// TwinCAT 3 PLC project M1L1_PLC
// ProgramVersion: 3.1.4020.5
// libraries:
//   LCLS General, * (SLAC)
//   Tc2_MC2, * (Beckhoff Automation GmbH)
//   Tc2_SerialCom, * (Beckhoff Automation GmbH)
//   Tc2_Standard, * (Beckhoff Automation GmbH)
//   Tc2_System, * (Beckhoff Automation GmbH)
//   Tc2_Utilities, * (Beckhoff Automation GmbH)
//   Tc3_Module, * (Beckhoff Automation GmbH)
//   lcls-twincat-motion,1.1.0,SLAC
// project tree:
//   Common/POUs/Helpers/ FB_PI_E621_SerialDriver.TcPOU (not stored), FB_PI_E621_SerialTransaction.TcPOU (not stored)
//   DUTs/ ST_PiezoAxis.TcDUT (not stored)
//   GVLs/ GVL_SerialIO.TcGVL (not stored)
//   / PlcTask.TcTTO (not stored), serial_com.TcTTO (not stored)
//   POUs/ MAIN.TcPOU
//   POUs/Serial Comm/ PiezoSerial.TcPOU (not stored), P_Serial_Com.TcPOU (not stored)
// real-time tasks:
//   TASK PlcTask: cycle T#10ms, priority 20, ADS port 350
//   TASK serial_com: cycle T#10ms, priority 21, ADS port 351
// motion (NC):
//   TASK NC-Task 1 SAF: cycle T#2ms, priority 4, ADS port 501
//   TASK NC-Task 1 SVB: cycle T#10ms, priority 8, ADS port 511
//   AXIS y_up (id 6)
//     General: UnitName=um
//     Dynamic: Acceleration=5050, Deceleration=5050, Jerk=5100500, DelayTime=0.008
//     Velo: Maximum=500
//     OtherSettings: AllowMotionCmdToSlave=true
//     encoder EncType=29
//       EncPara: ScaleFactorNumerator=1, ScaleFactorDenominator=1000, MaxCount=#xffffffff, ReferenceSystem=1
//         Inc: RefSoftSyncMask=#x0000ffff
//     drive DrvType=24
//       DrvPara: Inverse=true
//         Analog: VeloReferenz=500
//         TimeComp: TaskDelayCycles=1
//     controller CtrType=3
//       CtrPara: PriorControlFactor=1
//         PosDiffControl: Range=50, Time=0.2
//         PID: PosTn=0.005, PosIOutputLimit=0.0001, PosDOutputLimit=0, PosIDisableWhenMoving=true, DeadBandPosition=0.001
//         Observer: BandWidth=20
//   AXIS y_dwn (id 7)
//     General: UnitName=um
//     Dynamic: Acceleration=5050, Deceleration=5050, Jerk=5100500, DelayTime=0.008
//     Velo: Maximum=500
//     OtherSettings: AllowMotionCmdToSlave=true
//     encoder EncType=29
//       EncPara: ScaleFactorNumerator=1, ScaleFactorDenominator=1000, MaxCount=#xffffffff, ReferenceSystem=1
//         Inc: RefSoftSyncMask=#x0000ffff
//     drive DrvType=24
//       DrvPara: Inverse=true
//         Analog: VeloReferenz=500
//         TimeComp: TaskDelayCycles=1
//     controller CtrType=3
//       CtrPara: PriorControlFactor=1
//         PosDiffControl: Range=50, Time=0.2
//         PID: PosTn=0.005, PosIOutputLimit=0.0001, PosDOutputLimit=0, PosIDisableWhenMoving=true, DeadBandPosition=0.001
//         Observer: BandWidth=20
//   AXIS x_up (id 8)
//     General: UnitName=um
//     Dynamic: AccelerationMaximum=1000, DecelerationMaximum=1000, Acceleration=1000, Deceleration=1000, Jerk=5000, DelayTime=0.008
//     Velo: Maximum=625
//     OtherSettings: AllowMotionCmdToSlave=true
//     encoder EncType=29
//       EncPara: ScaleFactorNumerator=1, ScaleFactorDenominator=1000, MaxCount=#xffffffff, ReferenceSystem=1
//         Inc: RefSoftSyncMask=#x0000ffff
//     drive DrvType=24
//       Analog: VeloReferenz=625
//       TimeComp: TaskDelayCycles=1
//     controller CtrType=3
//       CtrPara: PriorControlFactor=1
//         PosDiffControl: Range=75, Time=0.2
//         PID: PosTn=0.005, PosIOutputLimit=0.0001, PosDOutputLimit=0, PosIDisableWhenMoving=true, DeadBandPosition=0.001
//         Observer: BandWidth=20
//   AXIS x_dwn (id 9)
//     General: UnitName=um
//     Dynamic: AccelerationMaximum=1000, DecelerationMaximum=1000, Acceleration=1000, Deceleration=1000, Jerk=5000, DelayTime=0.008
//     Velo: Maximum=625
//     OtherSettings: AllowMotionCmdToSlave=true
//     encoder EncType=29
//       EncPara: ScaleFactorNumerator=1, ScaleFactorDenominator=1000, MaxCount=#xffffffff, ReferenceSystem=1
//         Inc: RefSoftSyncMask=#x0000ffff
//     drive DrvType=24
//       DrvPara: Inverse=true
//         Analog: VeloReferenz=625
//         TimeComp: TaskDelayCycles=1
//     controller CtrType=3
//       CtrPara: PriorControlFactor=1
//         PosDiffControl: Range=75, Time=0.2
//         PID: PosTn=0.005, PosIOutputLimit=0.0001, PosDOutputLimit=0, PosIDisableWhenMoving=true, DeadBandPosition=0.001
//         Observer: BandWidth=20
//   AXIS pitch (id 10)
//     General: UnitName=urad
//     Dynamic: Acceleration=64082, Deceleration=64082, Jerk=711156, DelayTime=0.008
//     Velo: Maximum=400
//     OtherSettings: AllowMotionCmdToSlave=true
//     encoder EncType=29
//       EncPara: ScaleFactorNumerator=0.00244, MaxCount=#xffffffff, ReferenceSystem=1
//         ActPosCorrection: Time=0.008
//         Inc: RefSoftSyncMask=#x0000ffff
//     drive DrvType=24
//       DrvPara: Inverse=true
//         Analog: VeloReferenz=420
//         TimeComp: TaskDelayCycles=1
//     controller CtrType=3
//       CtrPara: PriorControlFactor=1
//         PosDiffControl: Range=10, Time=0.2
//         PID: PosKp=9, PosTn=0.0006, PosTv=1.2e-05, PosIOutputLimit=0.0005, PosDOutputLimit=0.0035, AccKa=0.001, DeadBandPosition=0.001
//         Observer: BandWidth=20
// I/O:
//   DEVICE Device 1 (EtherCAT), AmsNetId 5.54.18.124.2.1
//     Term 1 (EK1200)
//   DEVICE Device 4 (EtherCAT), AmsNetId 5.54.18.124.5.1
//     Term 4 (EK1100) [EK1100 EtherCAT Coupler (2A E-Bus)]
//       Term 5 (EL9410) [EL9410 E-Bus Power Supplier  (Diagnostics)]
//       Term 6 (EL7047) - Yup
//       Term 7 (EL7047) - Ydwn
//       Term 8 (EL7047) - Xup
//       Term 9 (EL7047) - Xdwn
//       Term 10 (EL7047) - PitchCoarse
//       Term 11 (EL5042) - Y [EL5042 2Ch. BiSS-C Encoder]
//       Term 12 (EL5042) - X
//       Term 13 (EL5042) - Pitch
//       Term 14 (EL6001) - PitchFine [EL6001 Interface (RS232)]
//       Term 15 (EL3054) [EL3054 4Ch. Ana. Input 4-20mA]
//       Term 16 (EL3202-0010) [EL3202-0010 2Ch. Ana. Input PT100 (RTD), High Precision]
//       Term 17 (EL3202-0010) [EL3202-0010 2Ch. Ana. Input PT100 (RTD), High Precision]
//       Term 33 (EL1004) [EL1004 4Ch. Dig. Input 24V, 3ms]
//       Term 15 (EL9011)
// variable links:
//   Axes/pitch <-> Device 4 (EtherCAT)/Term 4 (EK1100)/Term 10 (EL7047) - PitchCoarse
//     Drive/Inputs/In/nState1 @bit 3 <-> STM Status/Status/Error
//     Drive/Inputs/In/nState1 @bit 7 <-> STM Status/Status/Motor stall
//     Drive/Inputs/In/nState1 @bit 5 <-> STM Status/Status/Moving negative
//     Drive/Inputs/In/nState1 @bit 4 <-> STM Status/Status/Moving positive
//     Drive/Inputs/In/nState1 @bit 1 <-> STM Status/Status/Ready
//     Drive/Inputs/In/nState1 <-> STM Status/Status/Ready to enable
//     Drive/Inputs/In/nState1 @bit 6 <-> STM Status/Status/Torque reduced
//     Drive/Inputs/In/nState1 @bit 2 <-> STM Status/Status/Warning
//     Drive/Inputs/In/nState2 @bit 3 <-> STM Status/Status/Digital input 1
//     Drive/Inputs/In/nState2 @bit 4 <-> STM Status/Status/Digital input 2
//     Drive/Inputs/In/nState2 @bit 5 <-> STM Status/Status/Sync error
//     Drive/Inputs/In/nState2 @bit 7 <-> STM Status/Status/TxPDO Toggle
//     Drive/Inputs/In/nState4 @bit 1 <-> WcState/InputToggle
//     Drive/Inputs/In/nState4 <-> WcState/WcState
//     Drive/Outputs/Out/nCtrl1 <-> STM Control/Control/Enable
//     Drive/Outputs/Out/nCtrl1 @bit 2 <-> STM Control/Control/Reduce torque
//     Drive/Outputs/Out/nCtrl1 @bit 1 <-> STM Control/Control/Reset
//     Drive/Outputs/Out/nCtrl2 @bit 3 <-> STM Control/Control/Digital output 1
//     Drive/Outputs/Out/nDataOut2[0] <-> STM Velocity/Velocity
//   Axes/pitch <-> Device 4 (EtherCAT)/Term 4 (EK1100)/Term 13 (EL5042) - Pitch
//     Enc/Inputs/In/nComState @bit 1 <-> WcState/InputToggle
//     Enc/Inputs/In/nComState <-> WcState/WcState
//     Enc/Inputs/In/nDataIn1 <-> FB Inputs Channel 1/Position
//     Enc/Inputs/In/nState1 @bit 12 <-> FB Inputs Channel 1/Status/Diag
//     Enc/Inputs/In/nState1 @bit 1 <-> FB Inputs Channel 1/Status/Error
//     Enc/Inputs/In/nState1 @bit 14 <-> FB Inputs Channel 1/Status/Input cycle counter
//     Enc/Inputs/In/nState1 @bit 2 <-> FB Inputs Channel 1/Status/Ready
//     Enc/Inputs/In/nState1 @bit 13 <-> FB Inputs Channel 1/Status/TxPDO State
//     Enc/Inputs/In/nState1 <-> FB Inputs Channel 1/Status/Warning
//   Axes/x_dwn <-> Device 4 (EtherCAT)/Term 4 (EK1100)/Term 12 (EL5042) - X
//     Enc/Inputs/In/nComState @bit 1 <-> WcState/InputToggle
//     Enc/Inputs/In/nComState <-> WcState/WcState
//     Enc/Inputs/In/nDataIn1 <-> FB Inputs Channel 2/Position
//     Enc/Inputs/In/nState1 @bit 12 <-> FB Inputs Channel 2/Status/Diag
//     Enc/Inputs/In/nState1 @bit 1 <-> FB Inputs Channel 2/Status/Error
//     Enc/Inputs/In/nState1 @bit 14 <-> FB Inputs Channel 2/Status/Input cycle counter
//     Enc/Inputs/In/nState1 @bit 2 <-> FB Inputs Channel 2/Status/Ready
//     Enc/Inputs/In/nState1 @bit 13 <-> FB Inputs Channel 2/Status/TxPDO State
//     Enc/Inputs/In/nState1 <-> FB Inputs Channel 2/Status/Warning
//   Axes/x_dwn <-> Device 4 (EtherCAT)/Term 4 (EK1100)/Term 9 (EL7047) - Xdwn
//     Drive/Inputs/In/nState1 @bit 3 <-> STM Status/Status/Error
//     Drive/Inputs/In/nState1 @bit 7 <-> STM Status/Status/Motor stall
//     Drive/Inputs/In/nState1 @bit 5 <-> STM Status/Status/Moving negative
//     Drive/Inputs/In/nState1 @bit 4 <-> STM Status/Status/Moving positive
//     Drive/Inputs/In/nState1 @bit 1 <-> STM Status/Status/Ready
//     Drive/Inputs/In/nState1 <-> STM Status/Status/Ready to enable
//     Drive/Inputs/In/nState1 @bit 6 <-> STM Status/Status/Torque reduced
//     Drive/Inputs/In/nState1 @bit 2 <-> STM Status/Status/Warning
//     Drive/Inputs/In/nState2 @bit 3 <-> STM Status/Status/Digital input 1
//     Drive/Inputs/In/nState2 @bit 4 <-> STM Status/Status/Digital input 2
//     Drive/Inputs/In/nState2 @bit 5 <-> STM Status/Status/Sync error
//     Drive/Inputs/In/nState2 @bit 7 <-> STM Status/Status/TxPDO Toggle
//     Drive/Inputs/In/nState4 @bit 1 <-> WcState/InputToggle
//     Drive/Inputs/In/nState4 <-> WcState/WcState
//     Drive/Outputs/Out/nCtrl1 <-> STM Control/Control/Enable
//     Drive/Outputs/Out/nCtrl1 @bit 2 <-> STM Control/Control/Reduce torque
//     Drive/Outputs/Out/nCtrl1 @bit 1 <-> STM Control/Control/Reset
//     Drive/Outputs/Out/nCtrl2 @bit 3 <-> STM Control/Control/Digital output 1
//     Drive/Outputs/Out/nDataOut2[0] <-> STM Velocity/Velocity
//   Axes/x_up <-> Device 4 (EtherCAT)/Term 4 (EK1100)/Term 12 (EL5042) - X
//     Enc/Inputs/In/nComState @bit 1 <-> WcState/InputToggle
//     Enc/Inputs/In/nComState <-> WcState/WcState
//     Enc/Inputs/In/nDataIn1 <-> FB Inputs Channel 1/Position
//     Enc/Inputs/In/nState1 @bit 12 <-> FB Inputs Channel 1/Status/Diag
//     Enc/Inputs/In/nState1 @bit 1 <-> FB Inputs Channel 1/Status/Error
//     Enc/Inputs/In/nState1 @bit 14 <-> FB Inputs Channel 1/Status/Input cycle counter
//     Enc/Inputs/In/nState1 @bit 2 <-> FB Inputs Channel 1/Status/Ready
//     Enc/Inputs/In/nState1 @bit 13 <-> FB Inputs Channel 1/Status/TxPDO State
//     Enc/Inputs/In/nState1 <-> FB Inputs Channel 1/Status/Warning
//   Axes/x_up <-> Device 4 (EtherCAT)/Term 4 (EK1100)/Term 8 (EL7047) - Xup
//     Drive/Inputs/In/nState1 @bit 3 <-> STM Status/Status/Error
//     Drive/Inputs/In/nState1 @bit 7 <-> STM Status/Status/Motor stall
//     Drive/Inputs/In/nState1 @bit 5 <-> STM Status/Status/Moving negative
//     Drive/Inputs/In/nState1 @bit 4 <-> STM Status/Status/Moving positive
//     Drive/Inputs/In/nState1 @bit 1 <-> STM Status/Status/Ready
//     Drive/Inputs/In/nState1 <-> STM Status/Status/Ready to enable
//     Drive/Inputs/In/nState1 @bit 6 <-> STM Status/Status/Torque reduced
//     Drive/Inputs/In/nState1 @bit 2 <-> STM Status/Status/Warning
//     Drive/Inputs/In/nState2 @bit 3 <-> STM Status/Status/Digital input 1
//     Drive/Inputs/In/nState2 @bit 4 <-> STM Status/Status/Digital input 2
//     Drive/Inputs/In/nState2 @bit 5 <-> STM Status/Status/Sync error
//     Drive/Inputs/In/nState2 @bit 7 <-> STM Status/Status/TxPDO Toggle
//     Drive/Inputs/In/nState4 @bit 1 <-> WcState/InputToggle
//     Drive/Inputs/In/nState4 <-> WcState/WcState
//     Drive/Outputs/Out/nCtrl1 <-> STM Control/Control/Enable
//     Drive/Outputs/Out/nCtrl1 @bit 2 <-> STM Control/Control/Reduce torque
//     Drive/Outputs/Out/nCtrl1 @bit 1 <-> STM Control/Control/Reset
//     Drive/Outputs/Out/nCtrl2 @bit 3 <-> STM Control/Control/Digital output 1
//     Drive/Outputs/Out/nDataOut2[0] <-> STM Velocity/Velocity
//   Axes/y_dwn <-> Device 4 (EtherCAT)/Term 4 (EK1100)/Term 11 (EL5042) - Y
//     Enc/Inputs/In/nComState @bit 1 <-> WcState/InputToggle
//     Enc/Inputs/In/nComState <-> WcState/WcState
//     Enc/Inputs/In/nDataIn1 <-> FB Inputs Channel 2/Position
//     Enc/Inputs/In/nState1 @bit 12 <-> FB Inputs Channel 2/Status/Diag
//     Enc/Inputs/In/nState1 @bit 1 <-> FB Inputs Channel 2/Status/Error
//     Enc/Inputs/In/nState1 @bit 14 <-> FB Inputs Channel 2/Status/Input cycle counter
//     Enc/Inputs/In/nState1 @bit 2 <-> FB Inputs Channel 2/Status/Ready
//     Enc/Inputs/In/nState1 @bit 13 <-> FB Inputs Channel 2/Status/TxPDO State
//     Enc/Inputs/In/nState1 <-> FB Inputs Channel 2/Status/Warning
//   Axes/y_dwn <-> Device 4 (EtherCAT)/Term 4 (EK1100)/Term 7 (EL7047) - Ydwn
//     Drive/Inputs/In/nState1 @bit 3 <-> STM Status/Status/Error
//     Drive/Inputs/In/nState1 @bit 7 <-> STM Status/Status/Motor stall
//     Drive/Inputs/In/nState1 @bit 5 <-> STM Status/Status/Moving negative
//     Drive/Inputs/In/nState1 @bit 4 <-> STM Status/Status/Moving positive
//     Drive/Inputs/In/nState1 @bit 1 <-> STM Status/Status/Ready
//     Drive/Inputs/In/nState1 <-> STM Status/Status/Ready to enable
//     Drive/Inputs/In/nState1 @bit 6 <-> STM Status/Status/Torque reduced
//     Drive/Inputs/In/nState1 @bit 2 <-> STM Status/Status/Warning
//     Drive/Inputs/In/nState2 @bit 3 <-> STM Status/Status/Digital input 1
//     Drive/Inputs/In/nState2 @bit 4 <-> STM Status/Status/Digital input 2
//     Drive/Inputs/In/nState2 @bit 5 <-> STM Status/Status/Sync error
//     Drive/Inputs/In/nState2 @bit 7 <-> STM Status/Status/TxPDO Toggle
//     Drive/Inputs/In/nState4 @bit 1 <-> WcState/InputToggle
//     Drive/Inputs/In/nState4 <-> WcState/WcState
//     Drive/Outputs/Out/nCtrl1 <-> STM Control/Control/Enable
//     Drive/Outputs/Out/nCtrl1 @bit 2 <-> STM Control/Control/Reduce torque
//     Drive/Outputs/Out/nCtrl1 @bit 1 <-> STM Control/Control/Reset
//     Drive/Outputs/Out/nCtrl2 @bit 3 <-> STM Control/Control/Digital output 1
//     Drive/Outputs/Out/nDataOut2[0] <-> STM Velocity/Velocity
//   Axes/y_up <-> Device 4 (EtherCAT)/Term 4 (EK1100)/Term 11 (EL5042) - Y
//     Enc/Inputs/In/nComState @bit 1 <-> WcState/InputToggle
//     Enc/Inputs/In/nComState <-> WcState/WcState
//     Enc/Inputs/In/nDataIn1 <-> FB Inputs Channel 1/Position
//     Enc/Inputs/In/nState1 @bit 12 <-> FB Inputs Channel 1/Status/Diag
//     Enc/Inputs/In/nState1 @bit 1 <-> FB Inputs Channel 1/Status/Error
//     Enc/Inputs/In/nState1 @bit 14 <-> FB Inputs Channel 1/Status/Input cycle counter
//     Enc/Inputs/In/nState1 @bit 2 <-> FB Inputs Channel 1/Status/Ready
//     Enc/Inputs/In/nState1 @bit 13 <-> FB Inputs Channel 1/Status/TxPDO State
//     Enc/Inputs/In/nState1 <-> FB Inputs Channel 1/Status/Warning
//   Axes/y_up <-> Device 4 (EtherCAT)/Term 4 (EK1100)/Term 6 (EL7047) - Yup
//     Drive/Inputs/In/nState1 @bit 3 <-> STM Status/Status/Error
//     Drive/Inputs/In/nState1 @bit 7 <-> STM Status/Status/Motor stall
//     Drive/Inputs/In/nState1 @bit 5 <-> STM Status/Status/Moving negative
//     Drive/Inputs/In/nState1 @bit 4 <-> STM Status/Status/Moving positive
//     Drive/Inputs/In/nState1 @bit 1 <-> STM Status/Status/Ready
//     Drive/Inputs/In/nState1 <-> STM Status/Status/Ready to enable
//     Drive/Inputs/In/nState1 @bit 6 <-> STM Status/Status/Torque reduced
//     Drive/Inputs/In/nState1 @bit 2 <-> STM Status/Status/Warning
//     Drive/Inputs/In/nState2 @bit 3 <-> STM Status/Status/Digital input 1
//     Drive/Inputs/In/nState2 @bit 4 <-> STM Status/Status/Digital input 2
//     Drive/Inputs/In/nState2 @bit 5 <-> STM Status/Status/Sync error
//     Drive/Inputs/In/nState2 @bit 7 <-> STM Status/Status/TxPDO Toggle
//     Drive/Inputs/In/nState4 @bit 1 <-> WcState/InputToggle
//     Drive/Inputs/In/nState4 <-> WcState/WcState
//     Drive/Outputs/Out/nCtrl1 <-> STM Control/Control/Enable
//     Drive/Outputs/Out/nCtrl1 @bit 2 <-> STM Control/Control/Reduce torque
//     Drive/Outputs/Out/nCtrl1 @bit 1 <-> STM Control/Control/Reset
//     Drive/Outputs/Out/nCtrl2 @bit 3 <-> STM Control/Control/Digital output 1
//     Drive/Outputs/Out/nDataOut2[0] <-> STM Velocity/Velocity
//   M1L1_PLC Instance <-> Device 4 (EtherCAT)/Term 4 (EK1100)/Term 10 (EL7047) - PitchCoarse
//     PlcTask Inputs/MAIN.M5.bLimitBackwardEnable <-> STM Status/Status/Digital input 2
//     PlcTask Inputs/MAIN.M5.bLimitForwardEnable <-> STM Status/Status/Digital input 1
//   M1L1_PLC Instance <-> Device 4 (EtherCAT)/Term 4 (EK1100)/Term 11 (EL5042) - Y
//     PlcTask Inputs/MAIN.y_dwn_enc/Count <-> FB Inputs Channel 2/Position
//     PlcTask Inputs/MAIN.y_up_enc/Count <-> FB Inputs Channel 1/Position
//   M1L1_PLC Instance <-> Device 4 (EtherCAT)/Term 4 (EK1100)/Term 12 (EL5042) - X
//     PlcTask Inputs/MAIN.x_dwn_enc/Count <-> FB Inputs Channel 2/Position
//     PlcTask Inputs/MAIN.x_up_enc/Count <-> FB Inputs Channel 1/Position
//   M1L1_PLC Instance <-> Device 4 (EtherCAT)/Term 4 (EK1100)/Term 33 (EL1004)
//     PlcTask Inputs/MAIN.stoEnable <-> Channel 1/Input
//   M1L1_PLC Instance <-> Device 4 (EtherCAT)/Term 4 (EK1100)/Term 6 (EL7047) - Yup
//     PlcTask Inputs/MAIN.M1.bLimitBackwardEnable <-> STM Status/Status/Digital input 2
//     PlcTask Inputs/MAIN.M1.bLimitForwardEnable <-> STM Status/Status/Digital input 1
//   M1L1_PLC Instance <-> Device 4 (EtherCAT)/Term 4 (EK1100)/Term 7 (EL7047) - Ydwn
//     PlcTask Inputs/MAIN.M2.bLimitBackwardEnable <-> STM Status/Status/Digital input 2
//     PlcTask Inputs/MAIN.M2.bLimitForwardEnable <-> STM Status/Status/Digital input 1
//   M1L1_PLC Instance <-> Device 4 (EtherCAT)/Term 4 (EK1100)/Term 8 (EL7047) - Xup
//     PlcTask Inputs/MAIN.M3.bLimitBackwardEnable <-> STM Status/Status/Digital input 2
//     PlcTask Inputs/MAIN.M3.bLimitForwardEnable <-> STM Status/Status/Digital input 1
//   M1L1_PLC Instance <-> Device 4 (EtherCAT)/Term 4 (EK1100)/Term 9 (EL7047) - Xdwn
//     PlcTask Inputs/MAIN.M4.bLimitBackwardEnable <-> STM Status/Status/Digital input 2
//     PlcTask Inputs/MAIN.M4.bLimitForwardEnable <-> STM Status/Status/Digital input 1
//   M1L1_PLC Instance <-> NC-Task 1 SAF/Axes/pitch
//     PlcTask Inputs/MAIN.M5.Axis.NcToPlc <-> Outputs/ToPlc
//     PlcTask Outputs/MAIN.M5.Axis.PlcToNc <-> Inputs/FromPlc
//   M1L1_PLC Instance <-> NC-Task 1 SAF/Axes/x_dwn
//     PlcTask Inputs/MAIN.M4.Axis.NcToPlc <-> Outputs/ToPlc
//     PlcTask Outputs/MAIN.M4.Axis.PlcToNc <-> Inputs/FromPlc
//   M1L1_PLC Instance <-> NC-Task 1 SAF/Axes/x_up
//     PlcTask Inputs/MAIN.M3.Axis.NcToPlc <-> Outputs/ToPlc
//     PlcTask Outputs/MAIN.M3.Axis.PlcToNc <-> Inputs/FromPlc
//   M1L1_PLC Instance <-> NC-Task 1 SAF/Axes/y_dwn
//     PlcTask Inputs/MAIN.M2.Axis.NcToPlc <-> Outputs/ToPlc
//     PlcTask Outputs/MAIN.M2.Axis.PlcToNc <-> Inputs/FromPlc
//   M1L1_PLC Instance <-> NC-Task 1 SAF/Axes/y_up
//     PlcTask Inputs/MAIN.M1.Axis.NcToPlc <-> Outputs/ToPlc
//     PlcTask Outputs/MAIN.M1.Axis.PlcToNc <-> Inputs/FromPlc

// ---- POUs/MAIN.TcPOU
PROGRAM MAIN
VAR
//	{attribute 'TcLinkTo' := '.bLimFwd:=TIIB[y_up]^STM Status^Status^Digital input 1; .bLimBwd:=TIIB[y_up]^STM Status^Status^Digital input 2; .bSTO:=TIIB[di]^Channel 1^Input'}	
	{attribute 'TcLinkTo':='.bLimFwd:=TIIB[y_up]^STM Status^Status^Digital input 1'}		
    M1: DUT_MotionStage:=(nCommand:=3); // Yup
//	{attribute 'TcLinkTo' := '.bLimFwd:=TIIB[y_dwn]^STM Status^Status^Digital input 1; .bLimBwd:=TIIB[y_dwn]^STM Status^Status^Digital input 2'}
	M2: DUT_MotionStage:=(nCommand:=3); // Ydwn
//	{attribute 'TcLinkTo' := '.bLimFwd:=TIIB[x_up]^STM Status^Status^Digital input 1; .bLimBwd:=TIIB[x_up]^STM Status^Status^Digital input 2'}	
	M3: DUT_MotionStage:=(nCommand:=3); // Xup
//	{attribute 'TcLinkTo' := '.bLimFwd:=TIIB[x_dwn]^STM Status^Status^Digital input 1; .bLimBwd:=TIIB[x_dwn]^STM Status^Status^Digital input 2'}
	M4: DUT_MotionStage:=(nCommand:=3); // Xdwn
//	{attribute 'TcLinkTo' := '.bLimFwd:=TIIB[pitch]^STM Status^Status^Digital input 1; .bLimBwd:=TIIB[pitch]^STM Status^Status^Digital input 2'}	
	M5: DUT_MotionStage:=(nCommand:=3); // PitchCoarse

	fbMotionStage_x_up, fbMotionStage_x_dwn, fbMotionStage_y_up, fbMotionStage_y_dwn, fbMotionStage_pitch : FB_MotionStage;

	stoEnable AT %I* : BOOL;
	{attribute 'TcLinkTo' := '.Count:=TIIB[1-x_up_2-x_dwn]^FB Inputs Channel 1^Position'}	
	x_up_enc  AT %I*: ST_RenishawAbsEnc;
	{attribute 'TcLinkTo' := '.Count:=TIIB[1-x_up_2-x_dwn]^FB Inputs Channel 2^Position'}
	x_dwn_enc  AT %I*: ST_RenishawAbsEnc;
	{attribute 'TcLinkTo' := '.Count:=TIIB[1-y_up_2-y_dwn]^FB Inputs Channel 1^Position'}	
	y_up_enc  AT %I*: ST_RenishawAbsEnc;
	{attribute 'TcLinkTo' := '.Count:=TIIB[1-y_up_2-y_dwn]^FB Inputs Channel 2^Position'}
	y_dwn_enc  AT %I*: ST_RenishawAbsEnc;

	// Auto coupling function block
	fbAutoCoupleX : FB_GantryAutoCoupling;
	fbAutoCoupleY : FB_GantryAutoCoupling;
	bExecuteCoupleX : BOOL;
	bExecuteCoupleY : BOOL;
	bExecuteDecoupleX : BOOL;
	bExecuteDecoupleY : BOOL;
	bGantryAlreadyCoupledX : BOOL;
	bGantryAlreadyCoupledY : BOOL;
	
	// Gantry variables
	nCurrGantryX : LINT;
	nCurrGantryY : LINT;
	nGantryTolX : LINT := 25000;
	nGantryTolY : LINT := 25000;

	// Add Some Encoder Readback and Storage:
	fbData : FB_LREALBuffer;
	bExecuteDataStorage : BOOL := TRUE;
	fbStats : FB_BasicStats;
	arrEncOutput : ARRAY [1..1000] OF LREAL;
	fEncMean : LREAL;
	fEncStDev : LREAL;
END_VAR

// M1K1
// Buttons to enable motors: write 0 to enable, 2 to disable
M1.nEnableMode; // Yup
M2.nEnableMode; // Ydwn
M3.nEnableMode; // Xup
M4.nEnableMode; // Xdwn
M5.nEnableMode; // PitchCoarse

// Encoder Reference Values: Taking from Axilon FAT
//M1K1 Ref Vals
y_up_enc.Ref := 30312000;
y_dwn_enc.Ref := 29600000; // Using values from Axilon FAT
x_up_enc.Ref := 19649910;
x_dwn_enc.Ref := 19609100;
 
// Gantry Differences to monitor
nCurrGantryY := ((ULINT_TO_LINT(y_up_enc.Count) - ULINT_TO_LINT(y_up_enc.Ref)) - (ULINT_TO_LINT(y_dwn_enc.Count) - ULINT_TO_LINT(y_dwn_enc.Ref)));
nCurrGantryX := ((ULINT_TO_LINT(x_up_enc.Count) - ULINT_TO_LINT(x_up_enc.Ref)) - (ULINT_TO_LINT(x_dwn_enc.Count) - ULINT_TO_LINT(x_dwn_enc.Ref)));

// E-stop
M1.bHardwareEnable := stoEnable;
M2.bHardwareEnable := stoEnable;
M3.bHardwareEnable := stoEnable;
M4.bHardwareEnable := stoEnable;
M5.bHardwareEnable := stoEnable;

// Start Autocoupling
fbAutoCoupleX(nGantryTol:=nGantryTolX, Master:=M3, MasterEnc:=x_up_enc, Slave:=M4,
	          SlaveEnc:=x_dwn_enc, bExecuteCouple:=bExecuteCoupleX,
              bExecuteDecouple:=bExecuteDecoupleX,
              bGantryAlreadyCoupled=>bGantryAlreadyCoupledX);

fbAutoCoupleY(nGantryTol:=nGantryTolY, Master:=M1, MasterEnc:=y_up_enc, Slave:=M2,
	          SlaveEnc:=y_dwn_enc, bExecuteCouple:=bExecuteCoupleY,
              bExecuteDecouple:=bExecuteDecoupleY,
			  bGantryAlreadyCoupled=>bGantryAlreadyCoupledY);

fbMotionStage_y_up  (stMotionStage:=M1);
fbMotionStage_y_dwn (stMotionStage:=M2);
fbMotionStage_x_up  (stMotionStage:=M3);
fbMotionStage_x_dwn (stMotionStage:=M4);
fbMotionStage_pitch (stMotionStage:=M5);

// Add Some Encoder Readback and Storage:
fbData(bExecute:=bExecuteDataStorage,
       fInput:=M5.stAxisStatus.fActPosition,
       arrOutput=>arrEncOutput);
fbStats(aSignal:=arrEncOutput,
	    bAlwaysCalc:=TRUE,
		fMean=>fEncMean,
		fStDev=>fEncStDev);

END_PROGRAM
